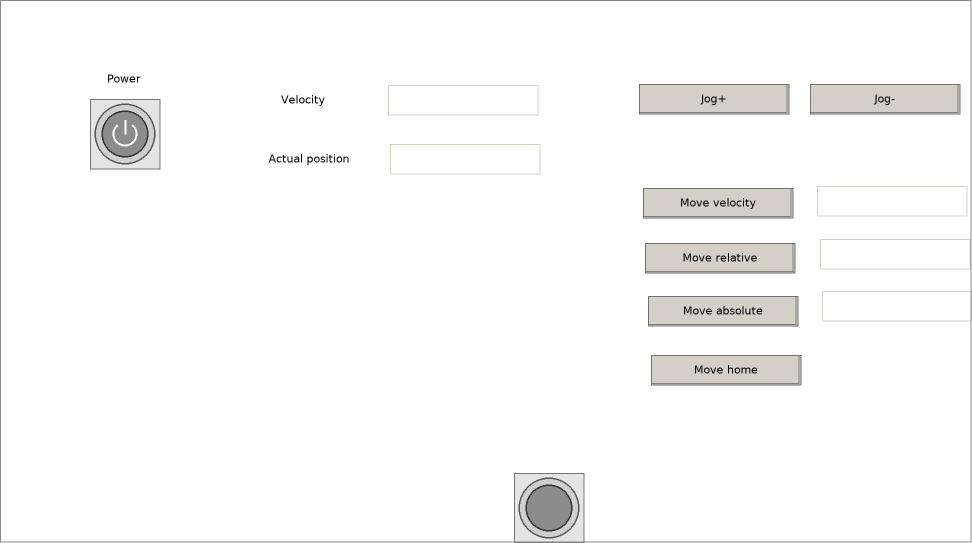
VISUALIZATION HMI  // 972x543
    PowerSwitch (90,99 70x70), variable: MAIN.AxisControl.McPowerEnable, behaviour: TOGGLE, style: Switch-PowerSwitch-Gray
    Label (49,64 150x30), "Power"
    Textfield (388,85 150x30)
    Textfield (390,144 150x30)
    Label (228,85 150x30), "Velocity"
    Label (234,144 150x30), "Actual position"
    Button (639,84 150x30), "Jog+"
    Button (810,84 150x30), "Jog-"
    Button (643,188 150x30), "Move velocity"
    Button (645,243 150x30), "Move relative"
    Button (648,296 150x30), "Move absolute"
    Button (651,355 150x30), "Move home"
    Textfield (817,186 150x30)
    Textfield (820,239 150x30)
    Textfield (822,291 150x30)
    PushSwitch (514,473 70x70), variable: MAIN.AxisControl.JogForward, behaviour: TOGGLE, style: Switch-PushSwitch-Gray
END_VISUALIZATION

(* stored: Version 1.1.0.1, ProductVersion 3.1.4024.13
   Visu HMI: Id {5cfdce4e-1e29-40f5-98cc-0ad19fd4d836} *)
